PROGRAM main
VAR
	Part_Sensor AT %IX0.0 : bool;
	Bin_Full_Light AT %QX0.0 : bool;
	Current_Count : int;
	R_TRIG0 : R_TRIG;
END_VAR
  VAR  (* added by the conversion: wires and edge detectors of the diagram *)
    _GT11_OUT : BOOL;
  END_VAR

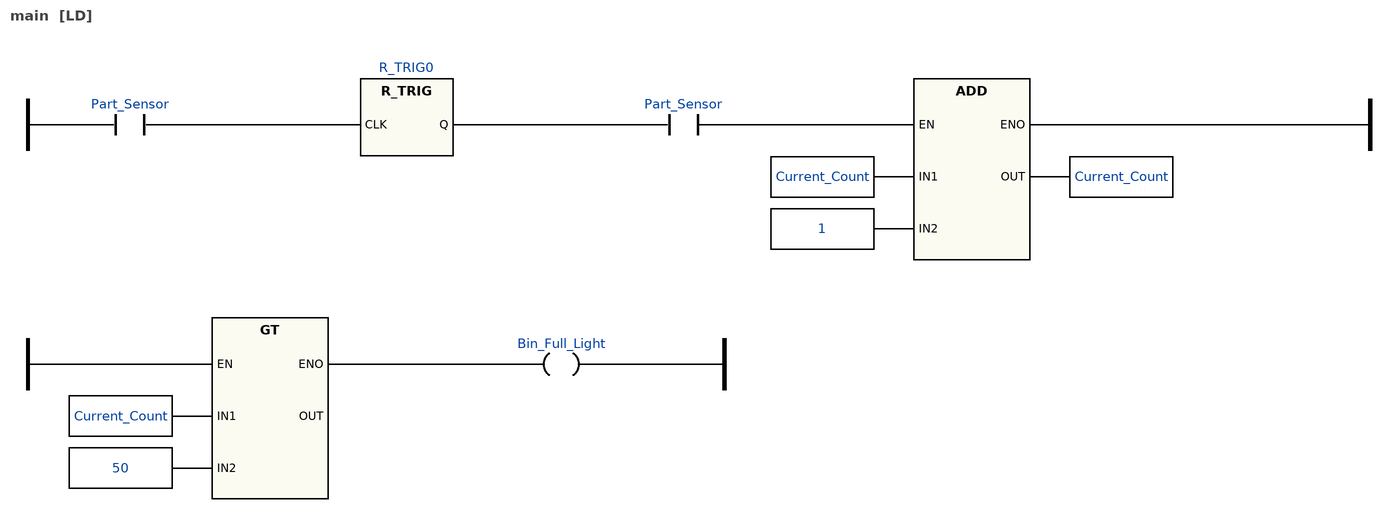
(* LD diagram, written out as Structured Text *)
R_TRIG0(CLK := Part_Sensor);
IF R_TRIG0.Q AND Part_Sensor THEN Current_Count := Current_Count + 1; END_IF;
_GT11_OUT := Current_Count > 50;
Bin_Full_Light := TRUE;
END_PROGRAM
